// Mitsubishi GX Works2 project: Automation2!   PLC: FX3G

// global labels: Global1
VAR_GLOBAL
  StartWorkDay AT X007 : BOOL;
  CurrentlyWorking AT Y007 : BOOL;
  TurnLightOff AT X005 : BOOL;
  NotEnoughProductDuring AT M50 : BOOL;
  NotEnoughProductStart AT M19 : BOOL;
  StartIceCreamMaking AT X001 : BOOL;
  YesNormalPetel AT M22 : BOOL;
  YesNormalLemon AT M23 : BOOL;
  CheckNormalGumi AT M24 : BOOL;
  ChoosePinuk AT M1 : BOOL;
  YesPinukPetel AT M25 : BOOL;
  YesPinukLemon AT M26 : BOOL;
  YesPinukGumi AT M27 : BOOL;
  ThereIsEnoughProductNormal AT M16 : BOOL;
  ThereIsEnoughProductPinuk AT M17 : BOOL;
  NotEnoughProductEnd AT M19 : BOOL;
  CheckL2LNormal AT M34 : BOOL;
  CheckP2PNormal AT M28 : BOOL;
  CheckL2PNormal AT M29 : BOOL;
  CheckH2PNormal AT M30 : BOOL;
  CheckP2PPinuk AT M31 : BOOL;
  CheckL2PPinuk AT M32 : BOOL;
  CheckH2PPinuk AT M33 : BOOL;
  CheckH2LNormal AT M35 : BOOL;
  CheckL2LPinuk AT M36 : BOOL;
  CheckH2LPinuk AT M37 : BOOL;
  SaveAnalog AT D8280 : INT;
END_VAR
VAR_GLOBAL CONSTANT
  MinPinuk : INT := 6;
  MaxNormal : INT := 5;
END_VAR
VAR_GLOBAL
  PetelInventory AT D1130 : REAL;
END_VAR
VAR_GLOBAL CONSTANT
  P2PNormalMin : REAL := 280;
  P2PPinukMin : REAL := 385;
END_VAR
VAR_GLOBAL
  LemonInventory AT D1140 : REAL;
END_VAR
VAR_GLOBAL CONSTANT
  L2PNormalMin : REAL := 35;
  L2LNormal : REAL := 420;
  L2LPinuk : REAL := 560;
  H2PNormal : REAL := 35;
END_VAR
VAR_GLOBAL
  HomerInventory AT D1150 : REAL;
END_VAR
VAR_GLOBAL CONSTANT
  H2PPinukl : REAL := 70;
  H2LNormal : REAL := 70;
  H2LPinuk : REAL := 140;
END_VAR
VAR_GLOBAL
  CheckP2PNormalEND AT M48 : BOOL;
  CheckP2PPinukEND AT M41 : BOOL;
  CheckL2PNormalEND AT M49 : BOOL;
  CheckL2PPinukEND AT M42 : BOOL;
  CheckL2LNormalEND AT M44 : BOOL;
  CheckL2LPinukEND AT M46 : BOOL;
  CheckH2PNormalEND AT M40 : BOOL;
  CheckH2PPinukEND AT M43 : BOOL;
  CheckH2LPinukEND AT M47 : BOOL;
  CheckH2LNormalEND AT M45 : BOOL;
  InputPetel AT D1100 : REAL;
  InputLemon AT D1102 : REAL;
  InputHomer AT D1104 : REAL;
  MakingTimer AT TC1 : BOOL;
END_VAR
VAR_GLOBAL CONSTANT
  DoneMaking : INT := 50;
END_VAR
VAR_GLOBAL
  Making AT TS1 : BOOL;
  CurrentlyMaking AT Y001 : BOOL;
  ChooseNormal AT M0 : BOOL;
END_VAR
VAR_GLOBAL CONSTANT
  L2PPinuk : REAL := 105;
  CheckGumiMin : REAL := 28;
END_VAR
VAR_GLOBAL
  GumiInventory AT D1160 : REAL;
END_VAR
VAR_GLOBAL CONSTANT
  MinusPetelNormal : REAL := 280;
  MinusLemonNormal : REAL := 455;
  MinusHomerNormal : REAL := 105;
  MinusGumiNormal : REAL := 28;
END_VAR
VAR_GLOBAL
  PackDone AT M60 : BOOL;
  InputGumi AT D1107 : REAL;
END_VAR
VAR_GLOBAL CONSTANT
  CheckGumiMinPinuk : REAL := 70;
  MinusPetelPinuk : REAL := 385;
  MinusLemonPinuk : REAL := 665;
  MinusHomerPinuk : REAL := 210;
  MinusGumiPinuk : REAL := 70;
END_VAR
VAR_GLOBAL
  YesNormaPetel AT M23 : BOOL;
END_VAR
VAR_GLOBAL CONSTANT
  Zero : REAL;
END_VAR
VAR_GLOBAL
  StartCooling AT X002 : BOOL;
  PetelIceCreamContainer AT D1110 : REAL;
END_VAR
VAR_GLOBAL CONSTANT
  PetelIceCream : REAL := 350;
END_VAR
VAR_GLOBAL
  LemonIceCreamContainer AT D1190 : REAL;
END_VAR
VAR_GLOBAL CONSTANT
  LemonIceCreamN : REAL := 490;
  PetelIceCreamN : REAL := 350;
  PetelIceCreamP : REAL := 560;
  LemonIceCreamP : REAL := 700;
END_VAR
VAR_GLOBAL
  PetelCooling AT D1112 : REAL;
END_VAR
VAR_GLOBAL CONSTANT
  ZEROPetel : REAL;
END_VAR
VAR_GLOBAL
  LemonCooling AT D1113 : REAL;
END_VAR
VAR_GLOBAL CONSTANT
  ZEROLemon : REAL;
END_VAR
VAR_GLOBAL
  CoolingTimer AT TC2 : BOOL;
END_VAR
VAR_GLOBAL CONSTANT
  DoneCooling : INT := 80;
END_VAR
VAR_GLOBAL
  Temp AT X003 : BOOL;
  CoolingEnd AT TS2 : BOOL;
  CoolingProcess AT Y002 : BOOL;
END_VAR
VAR_GLOBAL CONSTANT
  DIVIDEnum : INT := 400;
END_VAR
VAR_GLOBAL
  myAnalog AT D7000 : INT;
  MixIceCream AT D1195 : REAL;
  MixEndNormal AT TS3 : BOOL;
  MixTimer AT TC3 : BOOL;
END_VAR
VAR_GLOBAL CONSTANT
  DoneMix : INT := 30;
END_VAR
VAR_GLOBAL
  onn AT M61 : BOOL;
  Flashing5 AT TC4 : BOOL;
END_VAR
VAR_GLOBAL CONSTANT
  FlashingTime : WORD := 5;
END_VAR
VAR_GLOBAL
  Light5 AT Y005 : BOOL;
  Flashing6 AT TC5 : BOOL;
  EndFlashing6 AT TS5 : BOOL;
  Light6 AT Y006 : BOOL;
END_VAR
VAR_GLOBAL CONSTANT
  DoneMixPinuk : INT := 50;
END_VAR
VAR_GLOBAL
  FlashingHelp AT M62 : BOOL;
  MixTimerr AT TC6 : BOOL;
  TimeIr AT TC8 : BOOL;
  MixEndPinuk AT TS6 : BOOL;
  StartPack AT X004 : BOOL;
  DoneSevenPack AT CS10 : BOOL;
  PackCon AT X000 : BOOL;
  ConNumber AT CC9 : BOOL;
END_VAR
VAR_GLOBAL CONSTANT
  ConPacked : INT := 1;
END_VAR
VAR_GLOBAL
  SevenCones AT CC10 : BOOL;
  OneConePacked AT CS9 : BOOL;
  ReadyConePack AT D1198 : INT;
END_VAR
VAR_GLOBAL CONSTANT
  AddSevenPack : INT := 1;
END_VAR
VAR_GLOBAL
  analogOutput AT D8282 : INT;
END_VAR
VAR_GLOBAL CONSTANT
  ConstDivide : INT := 40;
END_VAR
VAR_GLOBAL
  StartAnalogOutput AT M100 : BOOL;
  EndFlashing5 AT TS4 : BOOL;
  Packing AT Y004 : BOOL;
  CheckK AT M70 : BOOL;
END_VAR

// task Task_01 (event TRUE, interval 0, priority 31): POU_01

PROGRAM POU_01
VAR CONSTANT
  SevenPacked : INT := 7;
END_VAR
(* structured ladder/FBD written out as ST: instructions are called as NAME(EN, inputs, outputs); _pN, _eN, _tN stand for wires *)
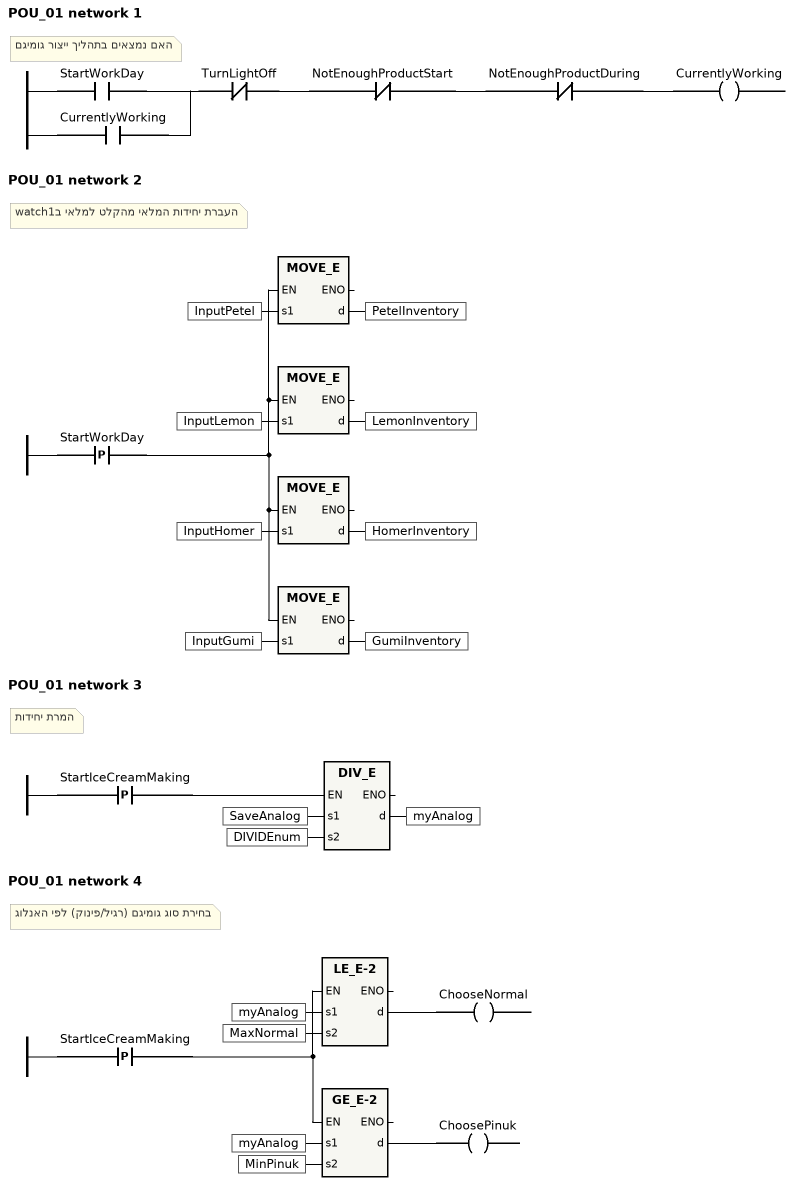
(* network 1 *)
(* האם נמצאים בתהליך ייצור גומיגם *)
CurrentlyWorking := (((StartWorkDay OR CurrentlyWorking) AND NOT TurnLightOff) AND NOT NotEnoughProductStart) AND NOT NotEnoughProductDuring;
(* network 2 *)
(* העברת יחידות המלאי מהקלט למלאי בwatch1 *)
_p1 := LDP(TRUE, StartWorkDay);
MOVE_E(_p1, InputPetel, PetelInventory);
MOVE_E(_p1, InputLemon, LemonInventory);
MOVE_E(_p1, InputHomer, HomerInventory);
MOVE_E(_p1, InputGumi, GumiInventory);
(* network 3 *)
(* המרת יחידות *)
DIV_E(LDP(TRUE, StartIceCreamMaking), SaveAnalog, DIVIDEnum, myAnalog);
(* network 4 *)
(* בחירת סוג גומיגם (רגיל/פינוק) לפי האנלוג *)
_p1 := LDP(TRUE, StartIceCreamMaking);
LE_E(_p1, myAnalog, MaxNormal, _t2);
ChooseNormal := _t2;
GE_E(_p1, myAnalog, MinPinuk, _t3);
ChoosePinuk := _t3;
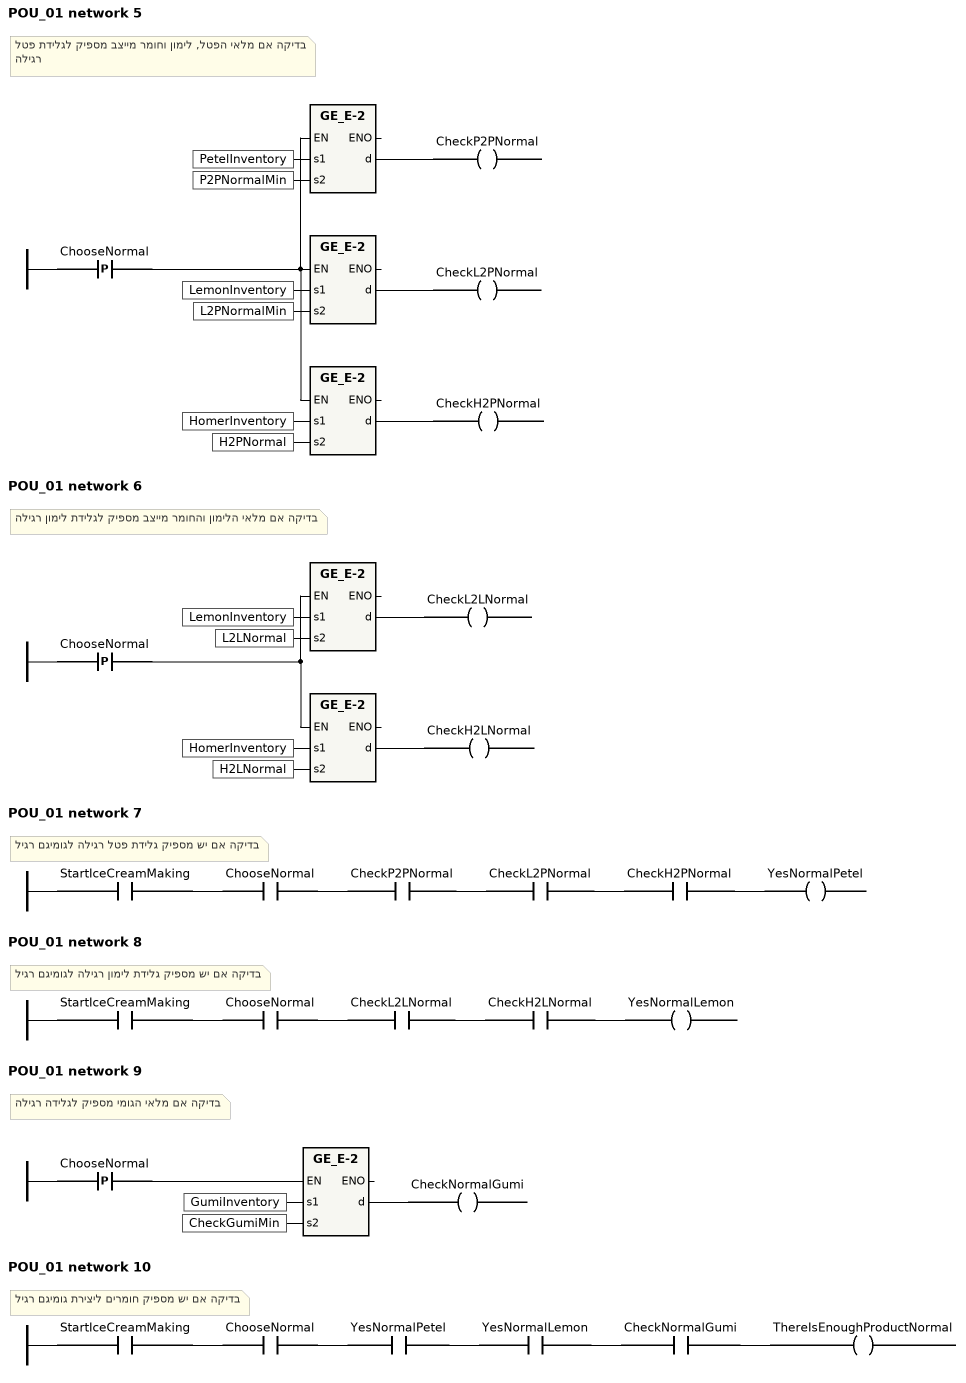
(* network 5 *)
(* בדיקה אם מלאי הפטל, לימון וחומר מייצב מספיק לגלידת פטל רגילה *)
_p1 := LDP(TRUE, ChooseNormal);
GE_E(_p1, PetelInventory, P2PNormalMin, _t2);
CheckP2PNormal := _t2;
GE_E(_p1, LemonInventory, L2PNormalMin, _t3);
CheckL2PNormal := _t3;
GE_E(_p1, HomerInventory, H2PNormal, _t4);
CheckH2PNormal := _t4;
(* network 6 *)
(* בדיקה אם מלאי הלימון והחומר מייצב מספיק לגלידת לימון רגילה *)
_p1 := LDP(TRUE, ChooseNormal);
GE_E(_p1, LemonInventory, L2LNormal, _t2);
CheckL2LNormal := _t2;
GE_E(_p1, HomerInventory, H2LNormal, _t3);
CheckH2LNormal := _t3;
(* network 7 *)
(* בדיקה אם יש מספיק גלידת פטל רגילה לגומיגם רגיל *)
YesNormalPetel := StartIceCreamMaking AND ChooseNormal AND CheckP2PNormal AND CheckL2PNormal AND CheckH2PNormal;
(* network 8 *)
(* בדיקה אם יש מספיק גלידת לימון רגילה לגומיגם רגיל *)
YesNormalLemon := StartIceCreamMaking AND ChooseNormal AND CheckL2LNormal AND CheckH2LNormal;
(* network 9 *)
(* בדיקה אם מלאי הגומי מספיק לגלידה רגילה *)
GE_E(LDP(TRUE, ChooseNormal), GumiInventory, CheckGumiMin, _t1);
CheckNormalGumi := _t1;
(* network 10 *)
(* בדיקה אם יש מספיק חומרים ליצירת גומיגם רגיל *)
ThereIsEnoughProductNormal := StartIceCreamMaking AND ChooseNormal AND YesNormalPetel AND YesNormalLemon AND CheckNormalGumi;
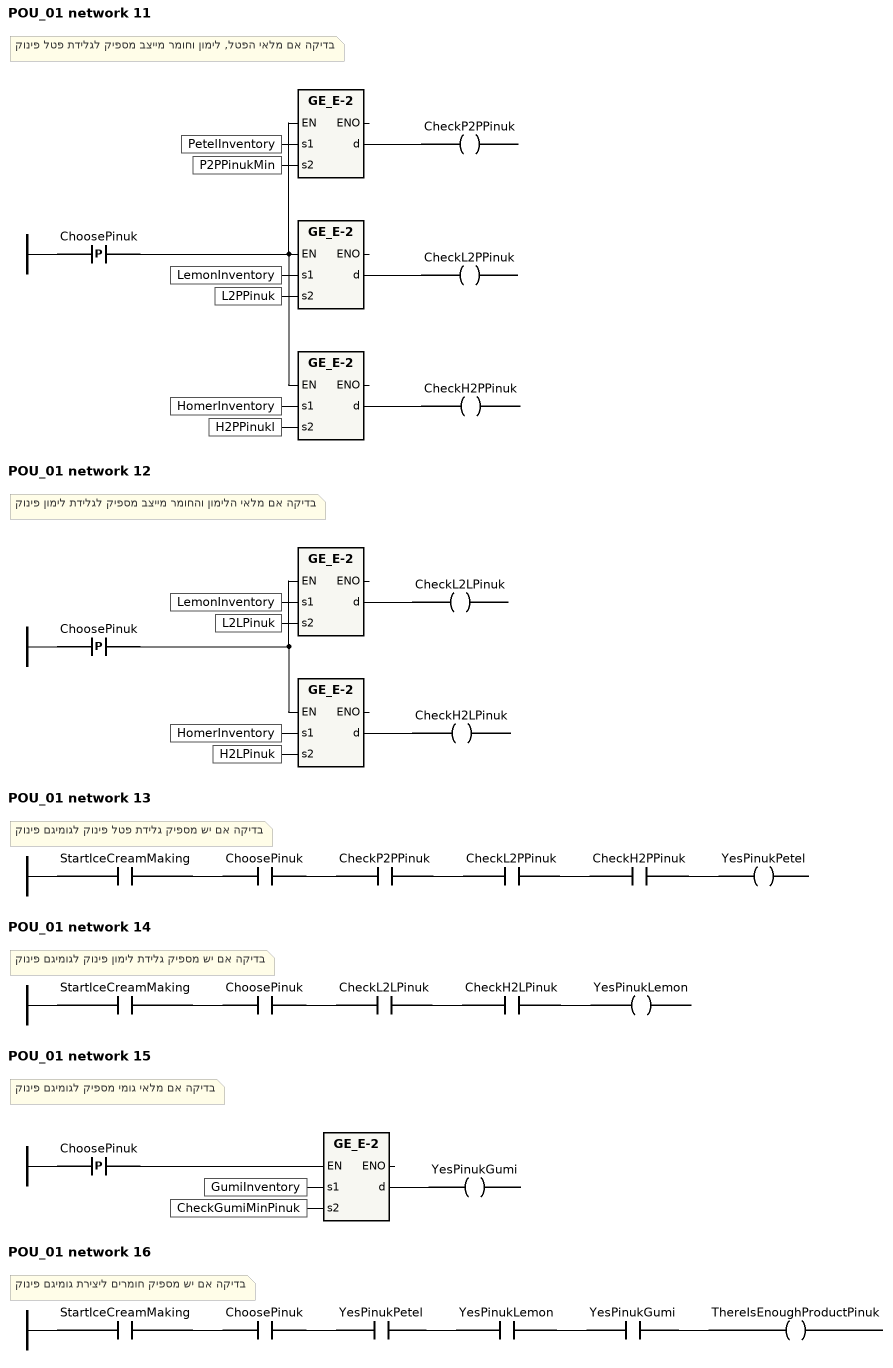
(* network 11 *)
(* בדיקה אם מלאי הפטל, לימון וחומר מייצב מספיק לגלידת פטל פינוק *)
_p1 := LDP(TRUE, ChoosePinuk);
GE_E(_p1, PetelInventory, P2PPinukMin, _t2);
CheckP2PPinuk := _t2;
GE_E(_p1, LemonInventory, L2PPinuk, _t3);
CheckL2PPinuk := _t3;
GE_E(_p1, HomerInventory, H2PPinukl, _t4);
CheckH2PPinuk := _t4;
(* network 12 *)
(* בדיקה אם מלאי הלימון והחומר מייצב מספיק לגלידת לימון פינוק *)
_p1 := LDP(TRUE, ChoosePinuk);
GE_E(_p1, LemonInventory, L2LPinuk, _t2);
CheckL2LPinuk := _t2;
GE_E(_p1, HomerInventory, H2LPinuk, _t3);
CheckH2LPinuk := _t3;
(* network 13 *)
(* בדיקה אם יש מספיק גלידת פטל פינוק לגומיגם פינוק *)
YesPinukPetel := StartIceCreamMaking AND ChoosePinuk AND CheckP2PPinuk AND CheckL2PPinuk AND CheckH2PPinuk;
(* network 14 *)
(* בדיקה אם יש מספיק גלידת לימון פינוק לגומיגם פינוק *)
YesPinukLemon := StartIceCreamMaking AND ChoosePinuk AND CheckL2LPinuk AND CheckH2LPinuk;
(* network 15 *)
(* בדיקה אם מלאי גומי מספיק לגומיגם פינוק *)
GE_E(LDP(TRUE, ChoosePinuk), GumiInventory, CheckGumiMinPinuk, _t1);
YesPinukGumi := _t1;
(* network 16 *)
(* בדיקה אם יש מספיק חומרים ליצירת גומיגם פינוק *)
ThereIsEnoughProductPinuk := StartIceCreamMaking AND ChoosePinuk AND YesPinukPetel AND YesPinukLemon AND YesPinukGumi;
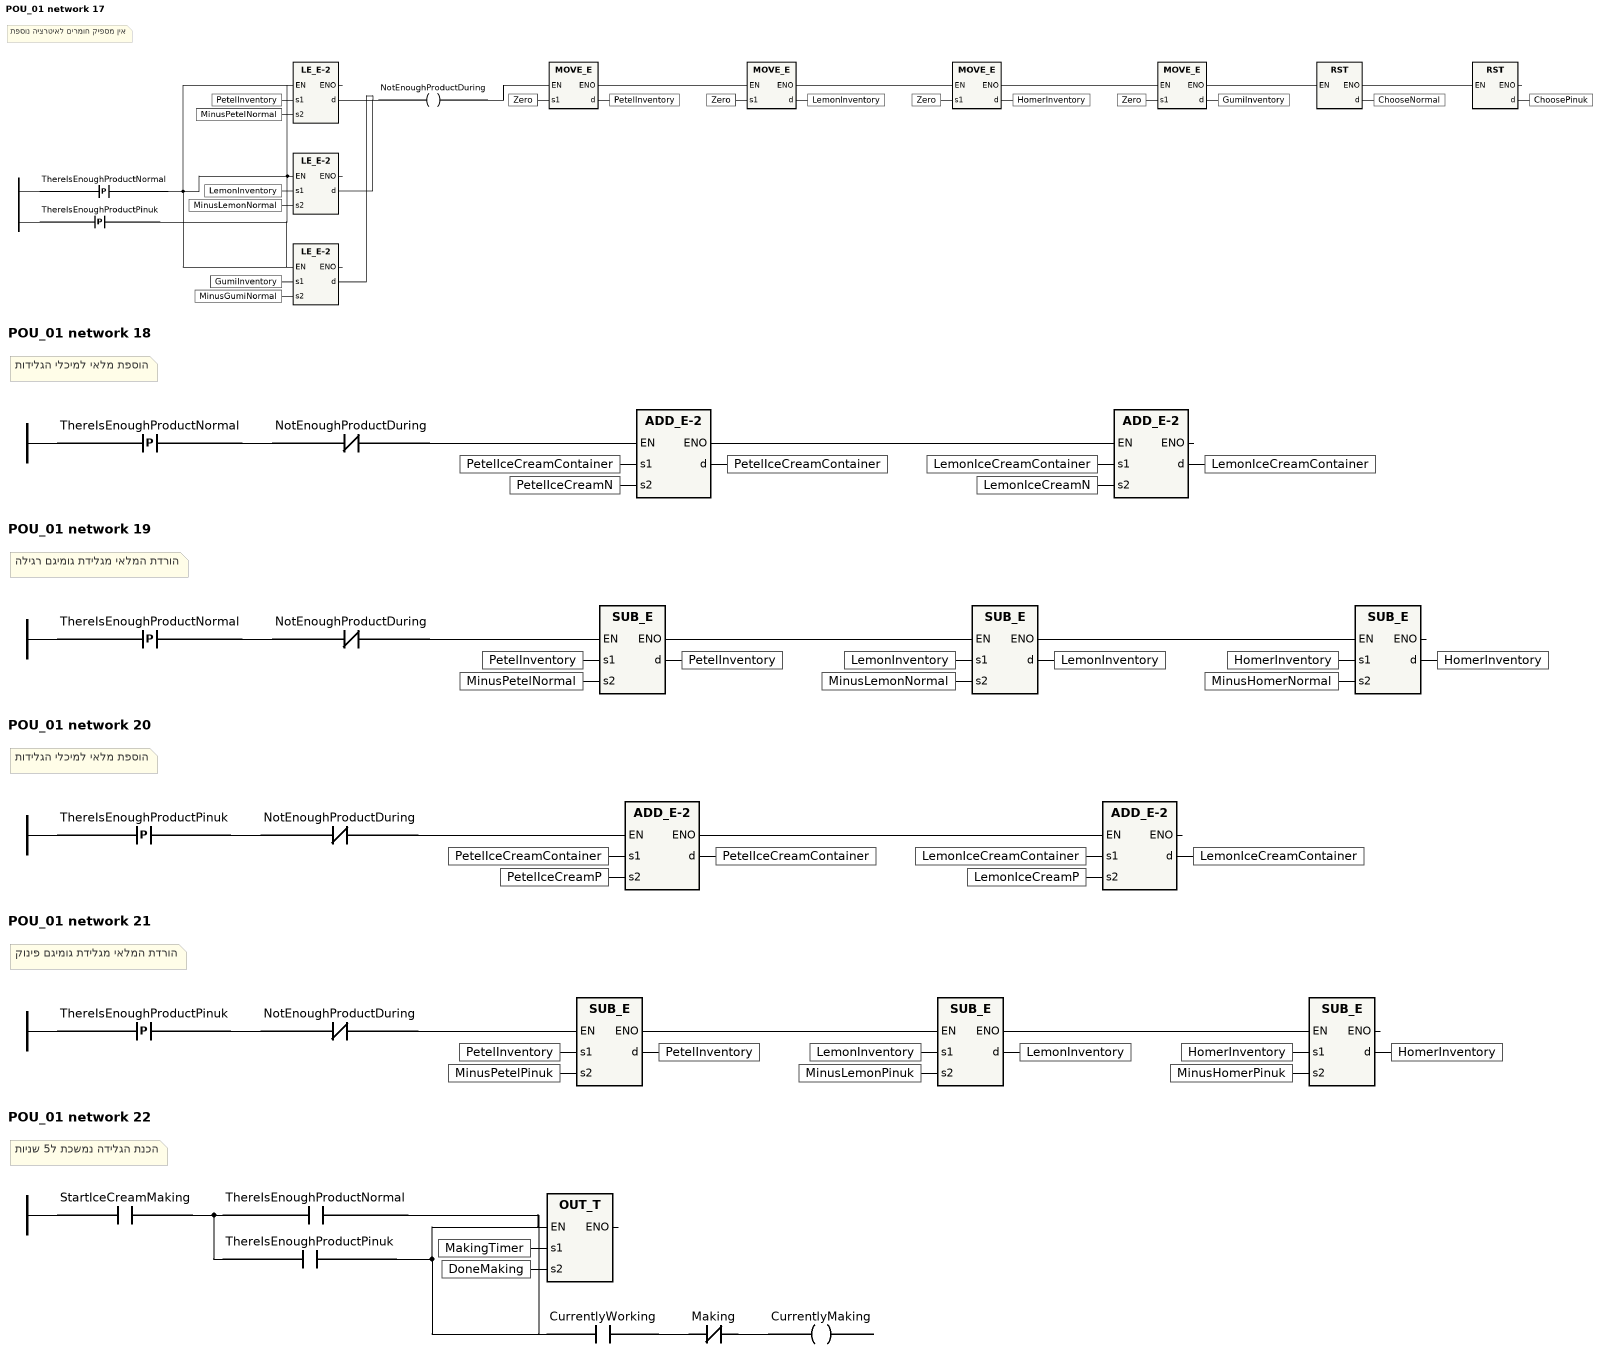
(* network 17 *)
(* אין מספיק חומרים לאיטרציה נוספת *)
_p1 := LDP(TRUE, ThereIsEnoughProductNormal) OR LDP(TRUE, ThereIsEnoughProductPinuk);
LE_E(_p1, PetelInventory, MinusPetelNormal, _t2);
LE_E(_p1, LemonInventory, MinusLemonNormal, _t3);
LE_E(_p1, GumiInventory, MinusGumiNormal, _t4);
_p5 := _t2 OR _t3 OR _t4;
NotEnoughProductDuring := _p5;
_e6 := MOVE_E(_p5, Zero, PetelInventory);
_e7 := MOVE_E(_e6, Zero, LemonInventory);
_e8 := MOVE_E(_e7, Zero, HomerInventory);
_e9 := MOVE_E(_e8, Zero, GumiInventory);
_e10 := RST(_e9, ChooseNormal);
RST(_e10, ChoosePinuk);
(* network 18 *)
(* הוספת מלאי למיכלי הגלידות *)
_e1 := ADD_E(LDP(TRUE, ThereIsEnoughProductNormal) AND NOT NotEnoughProductDuring, PetelIceCreamContainer, PetelIceCreamN, PetelIceCreamContainer);
ADD_E(_e1, LemonIceCreamContainer, LemonIceCreamN, LemonIceCreamContainer);
(* network 19 *)
(* הורדת המלאי מגלידת גומיגם רגילה *)
_e1 := SUB_E(LDP(TRUE, ThereIsEnoughProductNormal) AND NOT NotEnoughProductDuring, PetelInventory, MinusPetelNormal, PetelInventory);
_e2 := SUB_E(_e1, LemonInventory, MinusLemonNormal, LemonInventory);
SUB_E(_e2, HomerInventory, MinusHomerNormal, HomerInventory);
(* network 20 *)
(* הוספת מלאי למיכלי הגלידות *)
_e1 := ADD_E(LDP(TRUE, ThereIsEnoughProductPinuk) AND NOT NotEnoughProductDuring, PetelIceCreamContainer, PetelIceCreamP, PetelIceCreamContainer);
ADD_E(_e1, LemonIceCreamContainer, LemonIceCreamP, LemonIceCreamContainer);
(* network 21 *)
(* הורדת המלאי מגלידת גומיגם פינוק *)
_e1 := SUB_E(LDP(TRUE, ThereIsEnoughProductPinuk) AND NOT NotEnoughProductDuring, PetelInventory, MinusPetelPinuk, PetelInventory);
_e2 := SUB_E(_e1, LemonInventory, MinusLemonPinuk, LemonInventory);
SUB_E(_e2, HomerInventory, MinusHomerPinuk, HomerInventory);
(* network 22 *)
(* הכנת הגלידה נמשכת ל5 שניות *)
_p1 := (StartIceCreamMaking AND ThereIsEnoughProductNormal) OR (StartIceCreamMaking AND ThereIsEnoughProductPinuk);
CurrentlyMaking := _p1 AND CurrentlyWorking AND NOT Making;
OUT_T(_p1, MakingTimer, DoneMaking);
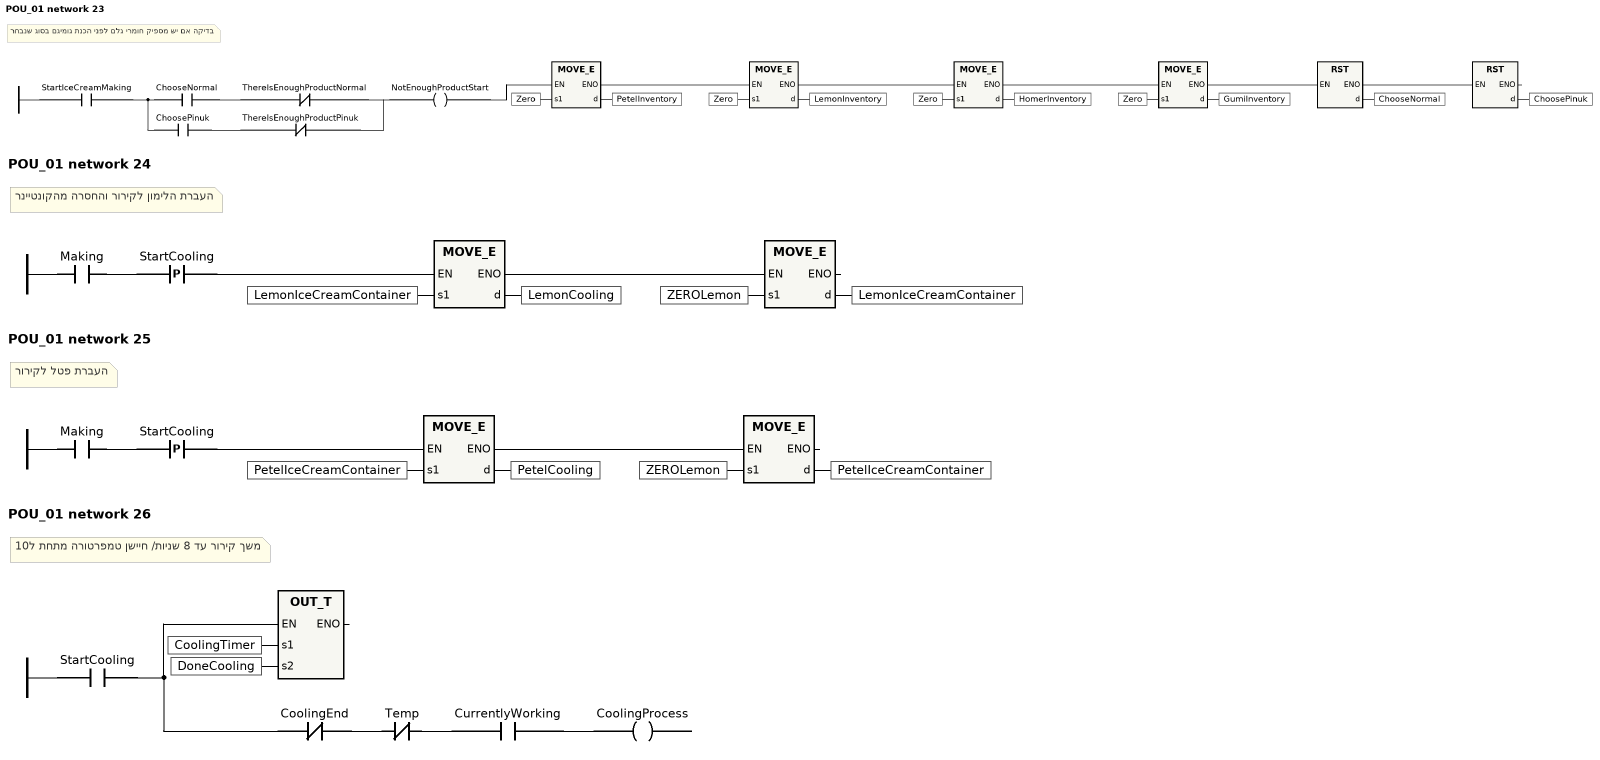
(* network 23 *)
(* בדיקה אם יש מספיק חומרי גלם לפני הכנת גומיגם בסוג שנבחר *)
_p1 := (StartIceCreamMaking AND ChooseNormal AND NOT ThereIsEnoughProductNormal) OR (StartIceCreamMaking AND ChoosePinuk AND NOT ThereIsEnoughProductPinuk);
NotEnoughProductStart := _p1;
_e2 := MOVE_E(_p1, Zero, PetelInventory);
_e3 := MOVE_E(_e2, Zero, LemonInventory);
_e4 := MOVE_E(_e3, Zero, HomerInventory);
_e5 := MOVE_E(_e4, Zero, GumiInventory);
_e6 := RST(_e5, ChooseNormal);
RST(_e6, ChoosePinuk);
(* network 24 *)
(* העברת הלימון לקירור והחסרה מהקונטיינר *)
_e1 := MOVE_E(Making AND LDP(TRUE, StartCooling), LemonIceCreamContainer, LemonCooling);
MOVE_E(_e1, ZEROLemon, LemonIceCreamContainer);
(* network 25 *)
(* העברת פטל לקירור *)
_e1 := MOVE_E(Making AND LDP(TRUE, StartCooling), PetelIceCreamContainer, PetelCooling);
MOVE_E(_e1, ZEROLemon, PetelIceCreamContainer);
(* network 26 *)
(* משך קירור עד 8 שניות/ חיישן טמפרטורה מתחת ל10 *)
OUT_T(StartCooling, CoolingTimer, DoneCooling);
CoolingProcess := StartCooling AND NOT CoolingEnd AND NOT Temp AND CurrentlyWorking;
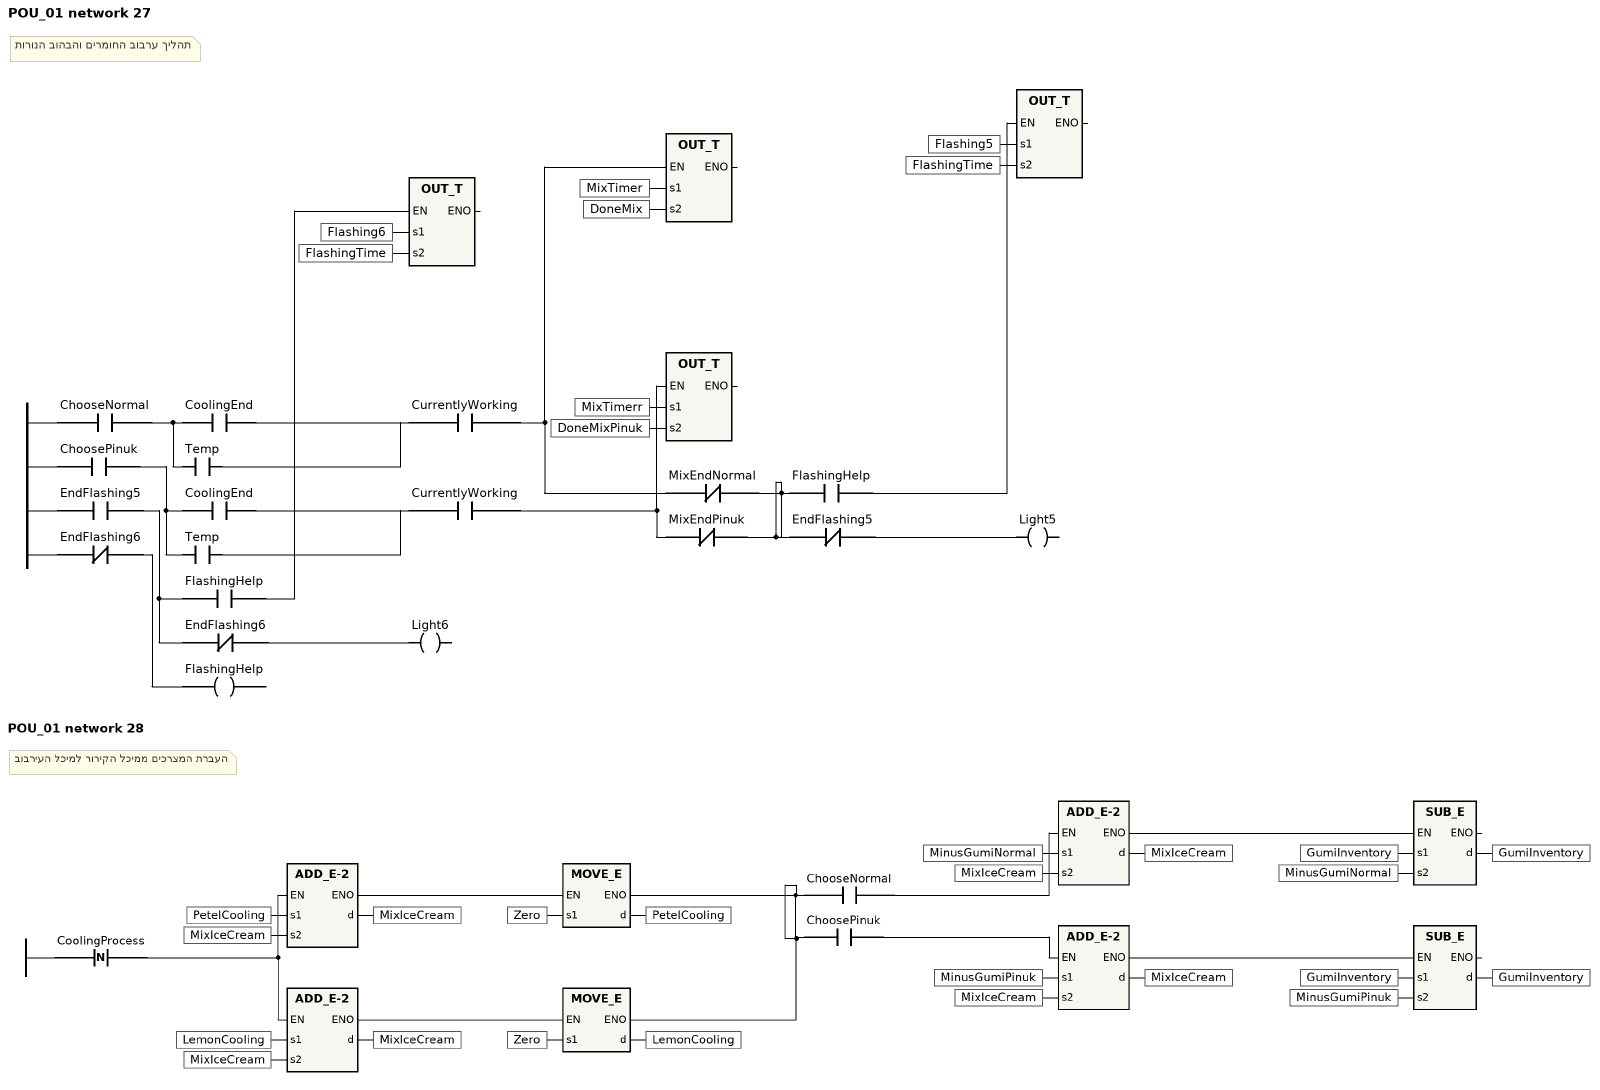
(* network 27 *)
(* תהליך ערבוב החומרים והבהוב הנורות *)
_p1 := ((ChooseNormal AND CoolingEnd) OR (ChooseNormal AND Temp)) AND CurrentlyWorking;
_p2 := ((ChoosePinuk AND CoolingEnd) OR (ChoosePinuk AND Temp)) AND CurrentlyWorking;
_p3 := (_p1 AND NOT MixEndNormal) OR (_p2 AND NOT MixEndPinuk);
OUT_T(_p3 AND FlashingHelp, Flashing5, FlashingTime);
Light5 := _p3 AND NOT EndFlashing5;
OUT_T(_p1, MixTimer, DoneMix);
OUT_T(_p2, MixTimerr, DoneMixPinuk);
OUT_T(EndFlashing5 AND FlashingHelp, Flashing6, FlashingTime);
Light6 := EndFlashing5 AND NOT EndFlashing6;
FlashingHelp := NOT EndFlashing6;
(* network 28 *)
(* העברת המצרכים ממיכל הקירור למיכל העירבוב *)
_p1 := LDF(TRUE, CoolingProcess);
_e2 := ADD_E(_p1, PetelCooling, MixIceCream, MixIceCream);
_e3 := MOVE_E(_e2, Zero, PetelCooling);
_e4 := ADD_E(_p1, LemonCooling, MixIceCream, MixIceCream);
_e5 := MOVE_E(_e4, Zero, LemonCooling);
_p6 := _e3 OR _e5;
_e7 := ADD_E(_p6 AND ChooseNormal, MinusGumiNormal, MixIceCream, MixIceCream);
SUB_E(_e7, GumiInventory, MinusGumiNormal, GumiInventory);
_e8 := ADD_E(_p6 AND ChoosePinuk, MinusGumiPinuk, MixIceCream, MixIceCream);
SUB_E(_e8, GumiInventory, MinusGumiPinuk, GumiInventory);
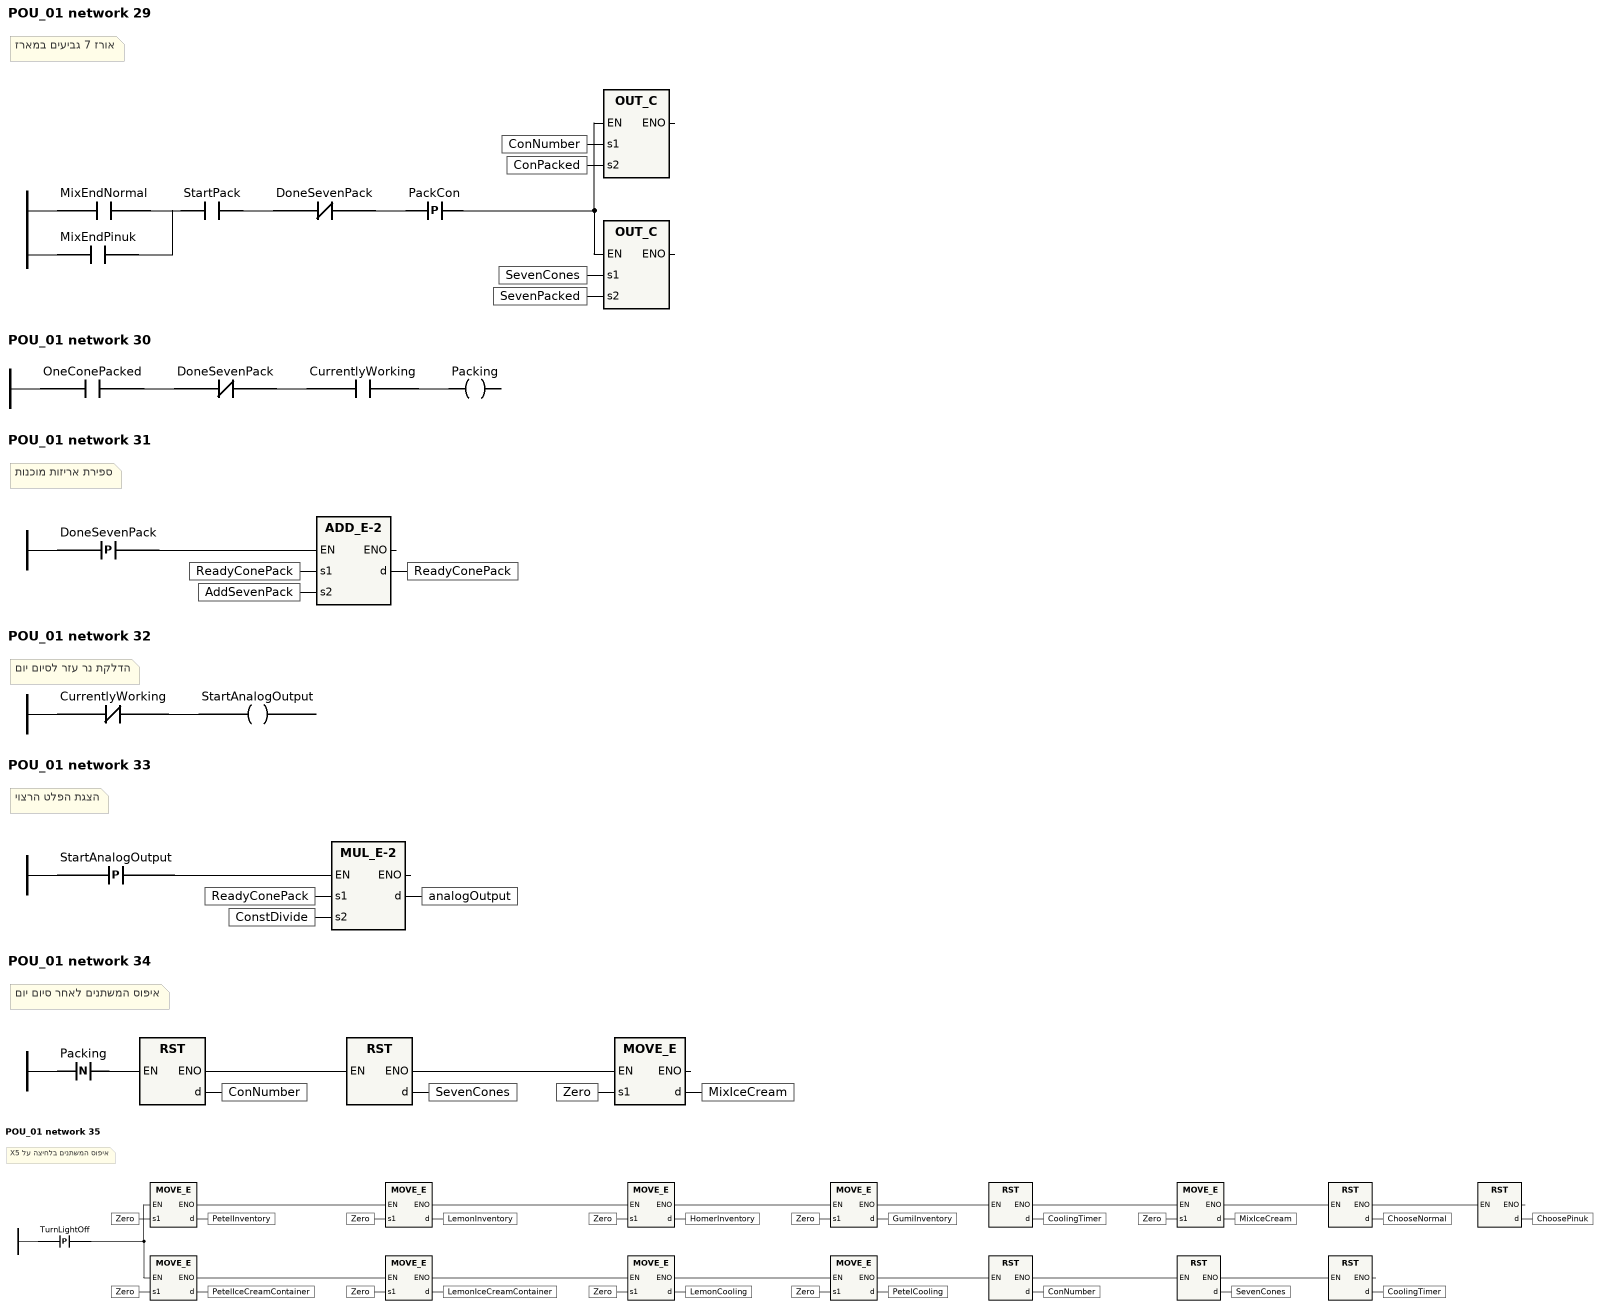
(* network 29 *)
(* אורז 7 גביעים במארז *)
_p1 := (((MixEndNormal OR MixEndPinuk) AND StartPack) AND NOT DoneSevenPack) AND LDP(TRUE, PackCon);
OUT_C(_p1, ConNumber, ConPacked);
OUT_C(_p1, SevenCones, SevenPacked);
(* network 30 *)
Packing := OneConePacked AND NOT DoneSevenPack AND CurrentlyWorking;
(* network 31 *)
(* ספירת אריזות מוכנות *)
ADD_E(LDP(TRUE, DoneSevenPack), ReadyConePack, AddSevenPack, ReadyConePack);
(* network 32 *)
(* הדלקת נר עזר לסיום יום *)
StartAnalogOutput := NOT CurrentlyWorking;
(* network 33 *)
(* הצגת הפלט הרצוי *)
MUL_E(LDP(TRUE, StartAnalogOutput), ReadyConePack, ConstDivide, analogOutput);
(* network 34 *)
(* איפוס המשתנים לאחר סיום יום *)
_e1 := RST(LDF(TRUE, Packing), ConNumber);
_e2 := RST(_e1, SevenCones);
MOVE_E(_e2, Zero, MixIceCream);
(* network 35 *)
(* איפוס המשתנים בלחיצה על X5 *)
_p1 := LDP(TRUE, TurnLightOff);
_e2 := MOVE_E(_p1, Zero, PetelInventory);
_e3 := MOVE_E(_e2, Zero, LemonInventory);
_e4 := MOVE_E(_e3, Zero, HomerInventory);
_e5 := MOVE_E(_e4, Zero, GumiInventory);
_e6 := RST(_e5, CoolingTimer);
_e7 := MOVE_E(_e6, Zero, MixIceCream);
_e8 := RST(_e7, ChooseNormal);
RST(_e8, ChoosePinuk);
_e9 := MOVE_E(_p1, Zero, PetelIceCreamContainer);
_e10 := MOVE_E(_e9, Zero, LemonIceCreamContainer);
_e11 := MOVE_E(_e10, Zero, LemonCooling);
_e12 := MOVE_E(_e11, Zero, PetelCooling);
_e13 := RST(_e12, ConNumber);
_e14 := RST(_e13, SevenCones);
RST(_e14, CoolingTimer);
END_PROGRAM
